FUNCTION_BLOCK FindFree
VAR_INPUT
	DrinkArray: ARRAY [1..25] OF Drinks;
	PalletArray: ARRAY [1..25] OF BOOL;
	TempDrink : Drinks;
	ErrorPosition : INT;
END_VAR
VAR_OUTPUT
	FreePosition : INT; 
END_VAR
VAR
	Counter : INT;
END_VAR

FreePosition := ErrorPosition;

FOR Counter:=1 TO 25 DO
 	IF NOT PalletArray[Counter] THEN
		IF DrinkArray[Counter] = TempDrink THEN
		FreePosition := Counter;
		END_IF
	END_IF
END_FOR

END_FUNCTION_BLOCK

(* stored: Version 1.1.0.1, ProductVersion 3.1.4022.12
   POU FindFree: Id {a9fbc3ff-d04d-4f8b-9fa0-8646871f6c2a}, SpecialFunc None *)
